Staubli VAL3: message.pgx

public program message(string& message[], num index)
// English IF message
begin
  // lenght of message
  //
  switch index
    case 0
      message="Desea editar:"
    break
    case 1
      message="< IF WIZARD >"
    break
    case 2
      message="Seleccione el tipo de condición a verificar"
    break
    case 3
      message="Seleccione la entrada"
    break
    case 4
      message="Seleccione la salida"
    break
    case 5
      message="Seleccione la entrada EMAP"
    break
    case 6
      message="Seleccione la manera de ejecutar la instrucción"
    break
    case 7
      message="Seleccione la instrucción a asociar a la :"
    break
    case 8
      message="Seleccione de la lista: "
    break
  endSwitch
end
